FUNCTION_BLOCK CFC_blinker
VAR_INPUT
	execute:BOOL;
	period: TIME := T#1S;
	duty: REAL := 0.5;
END_VAR
VAR_OUTPUT
	output:BOOL;
END_VAR
VAR
	delay: TON;
END_VAR
VAR // added by the converter: edge detectors and wires of the graphical bodies
    _w1 : ANY;
END_VAR

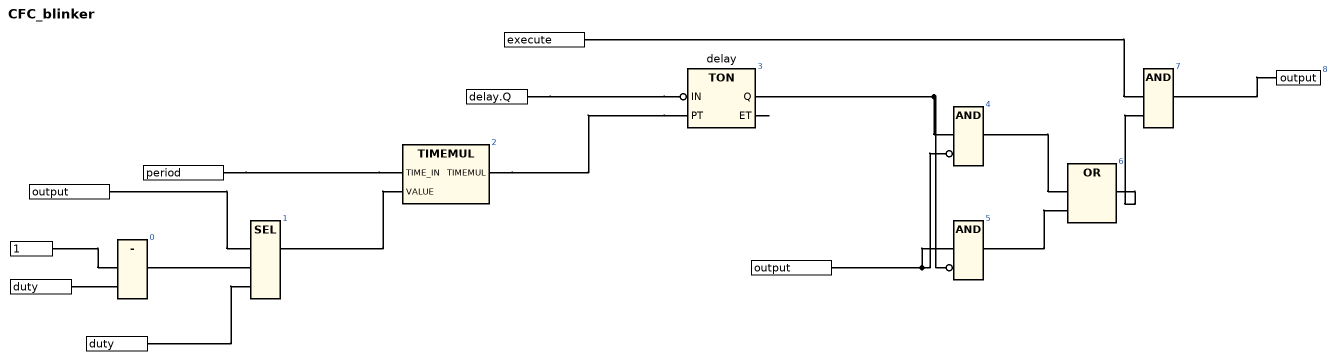
_w1 := TIMEMUL(TIME_IN := period, VALUE := SEL(output, 1 - duty, duty));
delay(IN := NOT delay.Q, PT := _w1); // TON
output := execute AND (delay.Q AND NOT output OR output AND NOT delay.Q);

END_FUNCTION_BLOCK

(* stored: Version 1.1.0.1, ProductVersion 3.1.4026.17
   POU CFC_blinker: Id {05c79bb3-e184-45a7-8159-56f2187c6d35}, SpecialFunc None *)
